// TIA Portal project "Programa_G10" (V18)

(* hardware
DEVICE "S71500/ET200MP station_1"  S7-1500 station
   slot 0: "Perfil soporte_0"  Rack  6ES7 590-1***0-0AA0
   slot 1: "PLC_1"  CPU 1516-3 PN/DP  6ES7 516-3AN01-0AB0  V2.1
      slot 3: "Display de la CPU_1"  6ES7591-1BA00-0AA0
   slot 2: "DI 32x24VDC HF_1"  DI 32x24VDC HF  6ES7 521-1BL00-0AB0  V2.1
   slot 3: "DQ 32x24VDC/0.5A HF_1"  DQ 32x24VDC/0.5A HF  6ES7 522-1BL01-0AB0  V1.0
   slot 4: "AI 8xU/I/RTD/TC ST_1"  AI 8xU/I/RTD/TC ST  6ES7 531-7KF00-0AB0  V2.1
   slot 5: "AQ 4xU/I ST_1"  AQ 4xU/I ST  6ES7 532-5HD00-0AB0  V2.1
*)

// ===== PLC "PLC_1"  CPU 1516-3 PN/DP =====

VAR_GLOBAL   // PLC tag table "Variables generales"
   "X10" AT %M0.0 : Bool;
   "X_PintadoModoCuadricula" AT %M0.1 : Bool;
   "X_PintadoModoNormal" AT %M0.2 : Bool;
   "ON" AT %E4.5 : Bool;
   "rearme" AT %E4.6 : Bool;
   "Seta_emergencia" AT %E4.7 : Bool;
   "X_Emer" AT %M0.3 : Bool;
END_VAR

VAR_GLOBAL   // PLC tag table "Estacion barnizado"
   "EST_BAR_SP_plat_omni" AT %E0.0 : Bool;
   "EST_BAR_pieza_debe_entrar" AT %E0.1 : Bool;
   "EST_BAR_SP_barnizadora_in" AT %E0.2 : Bool;
   "EST_BAR_SP_barnizadora_out" AT %E0.3 : Bool;
   "EST_BAR_SP_pickplace_grabado_in" AT %E0.4 : Bool;
   "EST_BAR_SP_pickplace_grabado_out" AT %E0.5 : Bool;
   "EST_BAR_SP_grabado" AT %E0.6 : Bool;
   "EST_BAR_Meter_Pieza" AT %A0.0 : Bool;
   "Temp_barnizadora" AT %T0 : Timer;
   "EST_BAR_Temp_ruedas_lim" AT %T1 : Timer;
   "EST_BAR_Temp_ruedas_std" AT %T2 : Timer;
   "EST_BAR_error_plat_omni" AT %A0.2 : Bool;
   "EST_BAR_emer_plat_omni" AT %A0.3 : Bool;
   "EST_BAR_stdby_plat_omni" AT %A0.4 : Bool;
   "EST_BAR_es_pieza" AT %E0.7 : Bool;
   "EST_BAR_es_cilindro" AT %E2.2 : Bool;
   "EST_BAR_es_tablero" AT %E1.1 : Bool;
   "EST_BAR_Temp_lim_pieza" AT %T3 : Timer;
   "EST_BAR_Temp_lim_cilindro" AT %T4 : Timer;
   "EST_BAR_Temp_lim_tablero" AT %T5 : Timer;
   "Barnizar_pieza" AT %A0.5 : Bool;
   "Barnizar_cilindro" AT %A0.6 : Bool;
   "Barnizar_tablero" AT %A0.7 : Bool;
   "EST_BAR_error_barnizadora" AT %A1.0 : Bool;
   "EST_BAR_emer_barnizadora" AT %A1.1 : Bool;
   "EST_BAR_stdby_barnizadora" AT %A1.2 : Bool;
   "EST_BAR_Temp_lim_pickplace_mov1" AT %T6 : Timer;
   "EST_BAR_Temp_lim_pickplace_mov2" AT %T7 : Timer;
   "EST_BAR_Temp_lim_pickplace_mov3" AT %T8 : Timer;
   "EST_BAR_Temp_lim_pickplace_mov4" AT %T9 : Timer;
   "EST_BAR_Temp_lim_pickplace_mov5" AT %T10 : Timer;
   "EST_BAR_pickplace_izq" AT %A1.3 : Bool;
   "EST_BAR_pickplace_coger" AT %A1.4 : Bool;
   "EST_BAR_pickplace_centro" AT %A1.5 : Bool;
   "EST_BAR_pickplace_soltar" AT %A1.6 : Bool;
   "EST_BAR_pickplace_ir_a_reposo" AT %A1.7 : Bool;
   "EST_BAR_pickplace_dcha" AT %A2.0 : Bool;
   "EST_BAR_pickplace_EnHome" AT %E1.2 : Bool;
   "EST_BAR_pickplace_EnIzq" AT %E1.3 : Bool;
   "EST_BAR_pickplace_EnCentro" AT %E1.4 : Bool;
   "EST_BAR_pickplace_EnDcha" AT %E1.5 : Bool;
   "EST_BAR_pickplace_pinza_ocupada" AT %E1.6 : Bool;
   "EST_BAR_pickplace_pinza_libre" AT %E1.7 : Bool;
   "EST_BAR_error_pickplace" AT %A2.1 : Bool;
   "EST_BAR_emer_pickplace" AT %A2.2 : Bool;
   "EST_BAR_stdby_pickplace" AT %A2.3 : Bool;
   "EST_BAR_Temp_lim_grabado" AT %T11 : Timer;
   "EST_BAR_Temp_std_grabado" AT %T12 : Timer;
   "EST_BAR_grabar" AT %A2.4 : Bool;
   "EST_BAR_error_grabado" AT %A2.5 : Bool;
   "EST_BAR_emer_grabado" AT %A2.6 : Bool;
   "EST_BAR_stdby_grabado" AT %A2.7 : Bool;
   "EST_BAR_grabado_terminado" AT %E2.3 : Bool;
END_VAR

VAR_GLOBAL   // PLC tag table "Estacion pintado"
   "EST_PIN_SP_plat_omni" AT %E2.0 : Bool;
   "EST_PINT_pieza_debe_entrar" AT %E2.1 : Bool;
   "EST_PIN_SP_pickplace_grabado_in" AT %E2.4 : Bool;
   "EST_PIN_SP_pickplace_grabado_out" AT %E2.5 : Bool;
   "EST_PIN_SP_pickplace_pintado_in" AT %E2.6 : Bool;
   "EST_PIN_SP_pickplace_pintado_out" AT %E2.7 : Bool;
   "EST_PIN_Temp_ruedas_lim" AT %T13 : Timer;
   "EST_PIN_Meter_Pieza" AT %A3.0 : Bool;
   "EST_PIN_error_plat_omni" AT %A3.1 : Bool;
   "EST_PIN_emer_plat_omni" AT %A3.2 : Bool;
   "EST_PIN_stdby_plat_omni" AT %A3.3 : Bool;
   "EST_PIN_SP_PiezaEnMesa" AT %E3.0 : Bool;
   "EST_PIN_SP_LaminaEnMesa" AT %E3.1 : Bool;
   "EST_PIN_SP_LaminaEnPosInicial" AT %E3.2 : Bool;
   "EST_PIN_Pintado_Terminado" AT %E3.3 : Bool;
   "EST_PIN_Hay_Tablero" AT %E3.4 : Bool;
   "EST_PIN_Temp_pintado_ModoLam" AT %T14 : Timer;
   "EST_PIN_Temp_pintado_ModoNormal" AT %T15 : Timer;
   "Pintar" AT %A3.4 : Bool;
   "EST_PIN_error_pintado" AT %A3.5 : Bool;
   "EST_PIN_emer_pintado" AT %A3.6 : Bool;
   "EST_PIN_stdby_pintado" AT %A3.7 : Bool;
   "EST_PIN_Temp_lim_pickplace_mov1" AT %T16 : Timer;
   "EST_PIN_Temp_lim_pickplace_mov2" AT %T17 : Timer;
   "EST_PIN_Temp_lim_pickplace_mov3" AT %T18 : Timer;
   "EST_PIN_Temp_lim_pickplace_mov4" AT %T19 : Timer;
   "EST_PIN_Temp_lim_pickplace_mov5" AT %T20 : Timer;
   "EST_PIN_pickplace_EnHome" AT %E3.5 : Bool;
   "EST_PIN_pickplace_EnIzq" AT %E3.6 : Bool;
   "EST_PIN_pickplace_EnCentro" AT %E3.7 : Bool;
   "EST_PIN_pickplace_EnDcha" AT %E4.0 : Bool;
   "EST_PIN_pickplace_pinza_ocupada" AT %E4.1 : Bool;
   "EST_PIN_pickplace_pinza_libre" AT %E4.2 : Bool;
   "EST_PIN_pickplace_izq" AT %A4.0 : Bool;
   "EST_PIN_pickplace_coger" AT %A4.1 : Bool;
   "EST_PIN_pickplace_centro" AT %A4.2 : Bool;
   "EST_PIN_pickplace_soltar" AT %A4.3 : Bool;
   "EST_PIN_pickplace_ir_a_reposo" AT %A4.4 : Bool;
   "EST_PIN_pickplace_dcha" AT %A4.5 : Bool;
   "EST_PIN_error_pickplace" AT %A4.6 : Bool;
   "EST_PIN_emer_pickplace" AT %A4.7 : Bool;
   "EST_PIN_stdby_pickplace" AT %A5.0 : Bool;
   "EST_PIN_SP_grabado" AT %E4.3 : Bool;
   "EST_PIN_grabado_terminado" AT %E4.4 : Bool;
   "EST_PIN_Temp_lim_grabado" AT %T21 : Timer;
   "EST_PIN_grabar" AT %A5.1 : Bool;
   "EST_PIN_error_grabado" AT %A5.2 : Bool;
   "EST_PIN_emer_grabado" AT %A5.3 : Bool;
   "EST_PIN_stdby_grabado" AT %A5.4 : Bool;
END_VAR

VAR_GLOBAL   // PLC tag table "Estacion secado"
   "EST_SEC_SP_plat_omni" AT %E1.0 : Bool;
   "EST_SEC_pieza_debe_entrar" AT %E5.0 : Bool;
   "EST_SEC_SP_secadora" AT %E5.1 : Bool;
   "EST_SEC_Meter_Pieza" AT %A5.6 : Bool;
   "EST_SEC_Temp_lim_ruedas" AT %T22 : Timer;
   "EST_SEC_error_plat_omni" AT %A5.7 : Bool;
   "EST_SEC_emer_plat_omni" AT %A6.0 : Bool;
   "EST_SEC_stdby_plat_omni" AT %A6.1 : Bool;
   "EST_SEC_secado_terminado" AT %E5.2 : Bool;
   "EST_SEC_Temp_lim_secado" AT %T23 : Timer;
   "Secar" AT %A6.2 : Bool;
   "EST_SEC_error_desecadora" AT %A6.3 : Bool;
   "EST_SEC_emer_desecadora" AT %A6.4 : Bool;
   "EST_SEC_stdby_desecadora" AT %A6.5 : Bool;
   "EST_SEC_SP_grabado" AT %E5.3 : Bool;
   "EST_SEC_grabado_terminado" AT %E5.4 : Bool;
   "EST_SEC_Temp_lim_grabado" AT %T24 : Timer;
   "EST_SEC_grabar" AT %A6.6 : Bool;
   "EST_SEC_error_grabado" AT %A6.7 : Bool;
   "EST_SEC_emer_grabado" AT %A7.0 : Bool;
   "EST_SEC_stdby_grabado" AT %A7.1 : Bool;
END_VAR

VAR_GLOBAL   // PLC tag table "Cinta"
   "vel_cinta_muestreada_bits" AT %EW4 : Int;
   "Temp_cinta" AT %T40 : Timer;
   "Error_cinta" AT %A10.0 : Bool;
   "Motor_cinta" AT %A10.1 : Bool;
   "velocidad_fuera_rango" AT %A10.2 : Bool;
END_VAR

DATA_BLOCK "Datos_produccion"   // DB1
{ S7_Optimized_Access := 'TRUE' }
VERSION : 0.1
   VAR
      t_lim_respuesta_lectura : S5Time := S5T#10s;
      t_lim_plat_omni : S5Time := S5T#60s;
      t_lim_barnizado : S5Time := S5T#10s;
      t_lim_secado : S5Time := S5T#60s;
      t_lim_pickandplace : S5Time := S5T#10s;
      t_lim_robotpintado : S5Time := S5T#10s;
      t_lim_grabado : S5Time := S5T#60s;
      t_lim_cinta : S5Time := S5T#10s;
      max_malas_lecturas : Word := 30;
      t_fugaz_21 : S5Time := S5T#1s;
      t_lim_pintado : S5Time;
      t_lim_barnizado_pieza : S5Time := S5T#30s;
      t_lim_barnizado_cilindro : S5Time := S5T#70s;
      t_lim_barnizado_tablero : S5Time := S5T#100s;
   END_VAR
BEGIN
END_DATA_BLOCK

// folder: Bloques de datos

DATA_BLOCK "Ruedas_omnidireccionales_DB_EST_BAR"   // DB2
{ S7_Optimized_Access := 'TRUE' }
VERSION : 0.1
// stored: InstanceOfName Ruedas_omnidireccionales
"Ruedas_omnidireccionales"
BEGIN
END_DATA_BLOCK

DATA_BLOCK "Maq_barnizado_DB"   // DB3
{ S7_Optimized_Access := 'TRUE' }
VERSION : 0.1
// stored: InstanceOfName Maq_barnizado
"Maq_barnizado"
BEGIN
END_DATA_BLOCK

DATA_BLOCK "Robot_pickandplace_DB_EST_BAR_1"   // DB4
{ S7_Optimized_Access := 'TRUE' }
VERSION : 0.1
// stored: InstanceOfName Robot_pickandplace
"Robot_pickandplace"
BEGIN
END_DATA_BLOCK

DATA_BLOCK "Maq_grabado_DB_EST_BAR"   // DB5
{ S7_Optimized_Access := 'TRUE' }
VERSION : 0.1
// stored: InstanceOfName Maq_grabado
"Maq_grabado"
BEGIN
END_DATA_BLOCK

DATA_BLOCK "Robot_pickandplace_DB_EST_BAR_2"   // DB6
{ S7_Optimized_Access := 'TRUE' }
VERSION : 0.1
// stored: InstanceOfName Robot_pickandplace
"Robot_pickandplace"
BEGIN
END_DATA_BLOCK

DATA_BLOCK "Ruedas_omnidireccionales_DB_EST_PINT"   // DB7
{ S7_Optimized_Access := 'TRUE' }
VERSION : 0.1
// stored: InstanceOfName Ruedas_omnidireccionales
"Ruedas_omnidireccionales"
BEGIN
END_DATA_BLOCK

DATA_BLOCK "Robot_pintado_DB"   // DB8
{ S7_Optimized_Access := 'TRUE' }
VERSION : 0.1
// stored: InstanceOfName Robot_pintado
"Robot_pintado"
BEGIN
END_DATA_BLOCK

DATA_BLOCK "Robot_pickandplace_DB_EST_PINT_1"   // DB9
{ S7_Optimized_Access := 'TRUE' }
VERSION : 0.1
// stored: InstanceOfName Robot_pickandplace
"Robot_pickandplace"
BEGIN
END_DATA_BLOCK

DATA_BLOCK "Maq_grabado_DB_EST_PINT"   // DB10
{ S7_Optimized_Access := 'TRUE' }
VERSION : 0.1
// stored: InstanceOfName Maq_grabado
"Maq_grabado"
BEGIN
END_DATA_BLOCK

DATA_BLOCK "Ruedas_omnidireccionales_DB_EST_SEC"   // DB11
{ S7_Optimized_Access := 'TRUE' }
VERSION : 0.1
// stored: InstanceOfName Ruedas_omnidireccionales
"Ruedas_omnidireccionales"
BEGIN
END_DATA_BLOCK

DATA_BLOCK "Maq_secado_DB"   // DB12
{ S7_Optimized_Access := 'TRUE' }
VERSION : 0.1
// stored: InstanceOfName Maq_secado
"Maq_secado"
BEGIN
END_DATA_BLOCK

DATA_BLOCK "Maq_grabado_DB_EST_SEC"   // DB13
{ S7_Optimized_Access := 'TRUE' }
VERSION : 0.1
// stored: InstanceOfName Maq_grabado
"Maq_grabado"
BEGIN
END_DATA_BLOCK

DATA_BLOCK "Cinta_DB"   // DB14
{ S7_Optimized_Access := 'TRUE' }
VERSION : 0.1
// stored: InstanceOfName Cinta
"Cinta"
BEGIN
END_DATA_BLOCK

// folder: Modos

DATA_BLOCK "Datos_ModoCuadricula"   // DB20
{ S7_Optimized_Access := 'TRUE' }
VERSION : 0.1
   VAR
      t_lim_pintado_ModoCuadricula : S5Time := S5T#100s;
   END_VAR
BEGIN
END_DATA_BLOCK

DATA_BLOCK "Datos_ModoNormal"   // DB21
{ S7_Optimized_Access := 'TRUE' }
VERSION : 0.1
   VAR
      t_lim_pintado_ModoNormal : S5Time := S5T#180s;
   END_VAR
BEGIN
END_DATA_BLOCK

// folder: (top level)

FUNCTION "Celda_barnizado_secado_pintado" : Void   // FC13, STL
{ S7_Optimized_Access := 'TRUE' }
VERSION : 0.1
BEGIN

REGION Network 1: Llamada a las estaciones
         CALL  "Estacion_barnizado";
         CALL  "Estacion_pintado";
         CALL  "Estacion_secado";
END_REGION

REGION Network 2: Llamada a la cinta

         CALL  "Cinta", "Cinta_DB"
         ( vel_cinta_bits        := "vel_cinta_muestreada_bits",
           t_lim_recuperacion    := "Datos_produccion".t_lim_cinta,
           Temp_lim              := "Temp_cinta",
           START                 := "ON",
           error_asincrono       := "Seta_emergencia",
           rearme                := "rearme",
           Act_motor             := "Motor_cinta",
           aviso_vel_fuera_rango := "Error_cinta"
         );
END_REGION

REGION Network 3: Llamada a las FC de emergencia y de modos
         CALL  "Emergencia";
         CALL  "Modos_pintado";
END_REGION
END_FUNCTION

ORGANIZATION_BLOCK "Main"   // OB1, STL, ProgramCycle
TITLE = "Main Program Sweep (Cycle)"
{ S7_Optimized_Access := 'TRUE' }
VERSION : 0.1
   VAR_INPUT
      Initial_Call : Bool;   // Initial call of this OB
      Remanence : Bool;   // =True, if remanent data are available
   END_VAR
BEGIN

REGION Network 1: Llamada a la celda de barnizado, secado y pintado
         CALL  "Celda_barnizado_secado_pintado";
END_REGION
END_ORGANIZATION_BLOCK

ORGANIZATION_BLOCK "Startup"   // OB100, STL, Startup
TITLE = "Complete Restart"
{ S7_Optimized_Access := 'TRUE' }
VERSION : 0.1
   VAR_INPUT
      LostRetentive : Bool;   // True if retentive data are lost
      LostRTC : Bool;   // True if date and time are lost
   END_VAR
BEGIN

REGION Network 1
         SET;
   //    S     "X0"
         S     "X10";
END_REGION
END_ORGANIZATION_BLOCK

// folder: Cinta

FUNCTION_BLOCK "Cinta"   // FB5, STL
{ S7_Optimized_Access := 'TRUE' }
VERSION : 0.1
   VAR_INPUT
      vel_cinta_bits : Int;
      t_lim_recuperacion : S5Time;
      Temp_lim : Timer;
      START : Bool;
      error_asincrono : Bool;
      rearme : Bool;
   END_VAR
   VAR_OUTPUT
      Act_motor : Bool;
      aviso_vel_fuera_rango : Bool;
   END_VAR
   VAR
      X1 : Bool;
      X2 : Bool;
      X_Err_Velocidad : Bool;
      X_Emer : Bool;
      bit_trabajo : Bool;
      vel_fuera_rango : Bool;
   END_VAR
   VAR_TEMP
      ret_val_scale : Word;
      vel_cinta_rpm : Real;
   END_VAR
BEGIN

REGION Network 1: Desconexión
         AN    #START;
         R     #bit_trabajo;
         R     #Act_motor;
         BEC;
END_REGION

REGION Network 2: Conexión
         A     #START;
         FP    #bit_trabajo;

         S     #X1;
         R     #X2;
         R     #X_Err_Velocidad;
END_REGION

REGION Network 3: Llamada a la función SCALE
         O     #X1;
         O     #X2;

         CALL  SCALE
         ( IN      := #vel_cinta_bits,
           HI_LIM  := 10000.0,
           LO_LIM  := 0.0,
           BIPOLAR := false,
           RET_VAL := #ret_val_scale,
           OUT     := #vel_cinta_rpm
         );
         O     #X1;
         O     #X2;
         A(;
         L     #ret_val_scale;
         L     W#16#0008;
         );
         ==I;
         =     #vel_fuera_rango;
END_REGION

REGION Network 4: X1 ->X2
         A     #X1;
         A     #vel_fuera_rango;
         S     #X2;
         R     #X1;
END_REGION

REGION Network 5: Configuración del temporizador
         A     #X2;
         L     #t_lim_recuperacion;
         SS    #Temp_lim;
END_REGION

REGION Network 6: X2-> X_Err_Cinta
         A     #X2;
         A     #Temp_lim;
         S     #X_Err_Velocidad;
         R     #X2;
END_REGION

REGION Network 7: X2 -> X1
         A     #X2;
         AN    #vel_fuera_rango;
         S     #X1;
         R     #X2;
         R     #Temp_lim;
         FR    #Temp_lim;
END_REGION

REGION Network 8: Tratamiento de X1
         A     #X1;
         S     #Act_motor;
END_REGION

REGION Network 9: Activación de X_Emer
         A     #error_asincrono;
         S     #X_Emer;
         R     #X2;
         R     #X_Err_Velocidad;
END_REGION

REGION Network 10: Tratamiento de X_Emer
         A     #X_Emer;
         R     #bit_trabajo;
         R     #aviso_vel_fuera_rango;
         R     #Act_motor;
         R     #Temp_lim;
         FR    #Temp_lim;
END_REGION

REGION Network 11: Rearme tras emergencia
         A     #X_Emer;
         A     #rearme;
         S     #X1;
         R     #X_Emer;
END_REGION

REGION Network 12: Tratamiento de X_Err_Cinta
         A     #X_Err_Velocidad;
         =     #aviso_vel_fuera_rango;
         A     #X_Err_Velocidad;
         R     #Act_motor;
END_REGION

REGION Network 13: Rearme tras error
         A     #X_Err_Velocidad;
         A     #rearme;
         S     #X1;
         R     #X_Err_Velocidad;
END_REGION
END_FUNCTION_BLOCK

// folder: Emergencia

FUNCTION "Emergencia" : Void   // FC3, STL
{ S7_Optimized_Access := 'TRUE' }
VERSION : 0.1
BEGIN

REGION Network 1: Tratamiento de X_EMER
         A     "Seta_emergencia";
         JCN   _TratamientoEmergencia;
   //LLAMADA A LA CINTA
         CALL  "Cinta", "Cinta_DB"
         ( vel_cinta_bits        := ,
           t_lim_recuperacion    := ,
           Temp_lim              := "Temp_cinta",
           START                 := ,
           error_asincrono       := TRUE,
           rearme                := ,
           Act_motor             := "Motor_cinta",
           aviso_vel_fuera_rango := "Error_cinta"
         );


   //LLAMADA A LAS MÁQUNAS Y ROBOTS DE LA ESTACION DE BARNIZADO
         CALL  "Ruedas_omnidireccionales", "Ruedas_omnidireccionales_DB_EST_BAR"
         ( START                          := ,
           SP_plataforma                  := ,
           evento_meter_pieza_en_estacion := ,
           pieza_metida                   := ,
           Temp_lim                       := "EST_BAR_Temp_ruedas_lim",
           tiempo_lim                     := ,
           EMER                           := true,
           rearme                         := ,
           Actuador                       := "EST_BAR_Meter_Pieza",
           aviso_error                    := "EST_BAR_error_plat_omni",
           aviso_emer                     := "EST_BAR_emer_plat_omni",
           aviso_stdby                    := "EST_BAR_stdby_plat_omni"
         );

         CALL  "Maq_barnizado", "Maq_barnizado_DB"
         ( START               := ,
           Sensor_inicio       := ,
           Sensor_fin          := ,
           evento_pieza        := ,
           evento_cilindro     := ,
           evento_tablero      := ,
           Temp_lim_pieza      := ,
           Temp_lim_cilindro   := "EST_BAR_Temp_lim_cilindro",
           Temp_lim_tablero    := "EST_BAR_Temp_lim_tablero",
           tiempo_lim_pieza    := ,
           tiempo_lim_cilindro := ,
           tiempo_lim_tablero  := ,
           EMER                := true,
           rearme              := ,
           Actuador_piezas     := "Barnizar_pieza",
           Actuador_cilindro   := "Barnizar_cilindro",
           Actuador_tablero    := "Barnizar_tablero",
           aviso_error_maq     := "EST_BAR_error_barnizadora",
           aviso_emer_maq      := "EST_BAR_emer_barnizadora",
           aviso_stdby         := "EST_BAR_stdby_barnizadora"
         );

         CALL  "Robot_pickandplace", "Robot_pickandplace_DB_EST_BAR_1"
         ( START             := ,
           emer              := true,
           rearme            := ,
           tiempo_lim        := ,
           Temp_lim_mov1     := "EST_BAR_Temp_lim_pickplace_mov1",
           Temp_lim_mov2     := "EST_BAR_Temp_lim_pickplace_mov2",
           Temp_lim_mov3     := "EST_BAR_Temp_lim_pickplace_mov3",
           Temp_lim_mov4     := "EST_BAR_Temp_lim_pickplace_mov4",
           Temp_lim_mov5     := "EST_BAR_Temp_lim_pickplace_mov5",
           Condicion_inicio  := ,
           Sensor_mov1       := ,
           Pinza_ocupada     := ,
           Sensor_mov3       := ,
           Pinza_libre       := ,
           Sensor_reposo     := ,
           Mov1              := "EST_BAR_pickplace_izq",
           Mov2              := "EST_BAR_pickplace_coger",
           Mov3              := "EST_BAR_pickplace_centro",
           Mov4              := "EST_BAR_pickplace_soltar",
           Mov5              := "EST_BAR_pickplace_ir_a_reposo",
           aviso_error_robot := "EST_BAR_error_pickplace",
           aviso_emer_robot  := "EST_BAR_emer_pickplace",
           aviso_stdby       := "EST_BAR_stdby_pickplace"
         );

         CALL  "Maq_grabado", "Maq_grabado_DB_EST_BAR"
         ( START                := ,
           Sensor_inicio        := ,
           maquina_ha_terminado := ,
           Temp_lim             := "EST_BAR_Temp_lim_grabado",
           tiempo_lim           := ,
           EMER                 := true,
           rearme               := ,
           Actuador             := "EST_BAR_grabar",
           aviso_error_maq      := "EST_BAR_error_grabado",
           aviso_emer_maq       := "EST_BAR_emer_grabado",
           aviso_stdby          := "EST_BAR_stdby_grabado",
           aviso_a_robot        :=
         );


         CALL  "Robot_pickandplace", "Robot_pickandplace_DB_EST_BAR_2"
         ( START             := ,
           emer              := true,
           rearme            := ,
           tiempo_lim        := ,
           Temp_lim_mov1     := "EST_BAR_Temp_lim_pickplace_mov1",
           Temp_lim_mov2     := "EST_BAR_Temp_lim_pickplace_mov2",
           Temp_lim_mov3     := "EST_BAR_Temp_lim_pickplace_mov3",
           Temp_lim_mov4     := "EST_BAR_Temp_lim_pickplace_mov4",
           Temp_lim_mov5     := "EST_BAR_Temp_lim_pickplace_mov5",
           Condicion_inicio  := ,
           Sensor_mov1       := ,
           Pinza_ocupada     := ,
           Sensor_mov3       := ,
           Pinza_libre       := ,
           Sensor_reposo     := ,
           Mov1              := "EST_BAR_pickplace_centro",
           Mov2              := "EST_BAR_pickplace_coger",
           Mov3              := "EST_BAR_pickplace_dcha",
           Mov4              := "EST_BAR_pickplace_soltar",
           Mov5              := "EST_BAR_pickplace_ir_a_reposo",
           aviso_error_robot := "EST_BAR_error_pickplace",
           aviso_emer_robot  := "EST_BAR_emer_pickplace",
           aviso_stdby       := "EST_BAR_stdby_pickplace"
         );



   //LLAMADA A LAS MAQUINAS Y ROBOTS DE LA ESTACION DE PINTADO

         CALL  "Ruedas_omnidireccionales", "Ruedas_omnidireccionales_DB_EST_PINT"
         ( START                          := ,
           SP_plataforma                  := ,
           evento_meter_pieza_en_estacion := ,
           pieza_metida                   := ,
           Temp_lim                       := "EST_PIN_Temp_ruedas_lim",
           tiempo_lim                     := ,
           EMER                           := TRUE,
           rearme                         := ,
           Actuador                       := "EST_PIN_Meter_Pieza",
           aviso_error                    := "EST_PIN_error_plat_omni",
           aviso_emer                     := "EST_PIN_emer_plat_omni",
           aviso_stdby                    := "EST_PIN_stdby_plat_omni"
         );

         CALL  "Robot_pickandplace", "Robot_pickandplace_DB_EST_PINT_1"
         ( START             := ,
           emer              := TRUE,
           rearme            := ,
           tiempo_lim        := ,
           Temp_lim_mov1     := "EST_PIN_Temp_lim_pickplace_mov1",
           Temp_lim_mov2     := "EST_PIN_Temp_lim_pickplace_mov2",
           Temp_lim_mov3     := "EST_PIN_Temp_lim_pickplace_mov3",
           Temp_lim_mov4     := "EST_PIN_Temp_lim_pickplace_mov4",
           Temp_lim_mov5     := "EST_PIN_Temp_lim_pickplace_mov5",
           Condicion_inicio  := ,
           Sensor_mov1       := ,
           Pinza_ocupada     := ,
           Sensor_mov3       := ,
           Pinza_libre       := ,
           Sensor_reposo     := ,
           Mov1              := "EST_PIN_pickplace_izq",
           Mov2              := "EST_PIN_pickplace_coger",
           Mov3              := "EST_PIN_pickplace_centro",
           Mov4              := "EST_PIN_pickplace_soltar",
           Mov5              := "EST_PIN_pickplace_ir_a_reposo",
           aviso_error_robot := "EST_PIN_error_pickplace",
           aviso_emer_robot  := "EST_PIN_emer_pickplace",
           aviso_stdby       := "EST_PIN_stdby_pickplace"
         );

         CALL  "Robot_pintado", "Robot_pintado_DB"
         ( SP_pieza                      := ,
           SP_lamina_mesa                := ,
           SP_lamina_pos_inicial         := ,
           robot_ha_terminado            := ,
           ModoLamina                    := ,
           ModoNormal                    := ,
           t_lim                         := ,
           EMER                          := true,
           rearme                        := ,
           START                         := ,
           Temp_lim_pintado_con_lam      := "EST_PIN_Temp_pintado_ModoLam",
           Temp_lim_pintado_sin_lam      := "EST_PIN_Temp_pintado_ModoNormal",
           Act_pintar                    := "Pintar",
           bde_tiempo                    := "EST_PIN_error_pintado",
           bit_stdby                     := "EST_PIN_stdby_pintado",
           bit_emer                      := "EST_PIN_emer_pintado",
           aviso_a_robot_lamina_a_mesa   := ,
           aviso_a_robot_lamina_a_origen :=
         );

         CALL  "Maq_grabado", "Maq_grabado_DB_EST_PINT"
         ( START                := ,
           Sensor_inicio        := ,
           maquina_ha_terminado := ,
           Temp_lim             := "EST_PIN_Temp_lim_grabado",
           tiempo_lim           := ,
           EMER                 := true,
           rearme               := ,
           Actuador             := "EST_PIN_grabar",
           aviso_error_maq      := "EST_PIN_error_grabado",
           aviso_emer_maq       := "EST_PIN_emer_grabado",
           aviso_stdby          := "EST_PIN_stdby_grabado",
           aviso_a_robot        :=
         );


   //LLAMADA A LAS MÁQUINAS Y ROBOTS DE LA ESTACIÓN DE SECADO

         CALL  "Ruedas_omnidireccionales", "Ruedas_omnidireccionales_DB_EST_SEC"
         ( START                          := ,
           SP_plataforma                  := ,
           evento_meter_pieza_en_estacion := ,
           pieza_metida                   := ,
           Temp_lim                       := "EST_SEC_Temp_lim_ruedas",
           tiempo_lim                     := ,
           EMER                           := true,
           rearme                         := ,
           Actuador                       := "EST_SEC_Meter_Pieza",
           aviso_error                    := "EST_SEC_error_plat_omni",
           aviso_emer                     := "EST_SEC_emer_plat_omni",
           aviso_stdby                    := "EST_SEC_stdby_plat_omni"
         );

         CALL  "Maq_secado", "Maq_secado_DB"
         ( START                := ,
           Sensor_inicio        := ,
           maquina_ha_terminado := ,
           Temp_lim             := "EST_SEC_Temp_lim_secado",
           tiempo_lim           := ,
           EMER                 := true,
           rearme               := ,
           Actuador             := "Secar",
           aviso_error_maq      := "EST_SEC_error_plat_omni",
           aviso_emer_maq       := "EST_SEC_emer_plat_omni",
           aviso_stdby          := "EST_SEC_stdby_plat_omni",
           aviso_a_robot        :=
         );

         CALL  "Maq_grabado", "Maq_grabado_DB_EST_SEC"
         ( START                := ,
           Sensor_inicio        := ,
           maquina_ha_terminado := ,
           Temp_lim             := "EST_SEC_Temp_lim_grabado",
           tiempo_lim           := ,
           EMER                 := true,
           rearme               := ,
           Actuador             := "EST_SEC_grabar",
           aviso_error_maq      := "EST_SEC_error_grabado",
           aviso_emer_maq       := "EST_SEC_emer_grabado",
           aviso_stdby          := "EST_SEC_stdby_grabado",
           aviso_a_robot        :=
         );


   _TratamientoEmergencia:NOP   0;
         A     "Seta_emergencia";
         R     "X_PintadoModoCuadricula";
         R     "X_PintadoModoNormal";

         BEC;
END_REGION

REGION Network 2: Rearme de la celda mediante el pulsador de rearme sin estar la seta activada.
         A     "X_Emer";
         A     "rearme";
         AN    "Seta_emergencia";
         S     "X10";
         R     "X_Emer";
END_REGION
END_FUNCTION

// folder: Estaciones

FUNCTION "Estacion_secado" : Void   // FC2, STL
{ S7_Optimized_Access := 'TRUE' }
VERSION : 0.1
   VAR_TEMP
      aviso_robot_recoger_pieza_secado : Bool;
      aviso_robot_recoger_pieza_grabado : Bool;
   END_VAR
BEGIN

REGION Network 1
         CALL  "Ruedas_omnidireccionales", "Ruedas_omnidireccionales_DB_EST_SEC"
         ( START                          := "ON",
           SP_plataforma                  := "EST_SEC_SP_plat_omni",
           evento_meter_pieza_en_estacion := "EST_SEC_pieza_debe_entrar",
           pieza_metida                   := "EST_SEC_SP_secadora",
           Temp_lim                       := "EST_SEC_Temp_lim_ruedas",
           tiempo_lim                     := "Datos_produccion".t_lim_plat_omni,
           EMER                           := false,
           rearme                         := "rearme",
           Actuador                       := "EST_SEC_Meter_Pieza",
           aviso_error                    := "EST_SEC_error_plat_omni",
           aviso_emer                     := "EST_SEC_emer_plat_omni",
           aviso_stdby                    := "EST_SEC_stdby_plat_omni"
         );

   //Llamada al pick and place para meter la pieza a la máquina de secado

         CALL  "Maq_secado", "Maq_secado_DB"
         ( START                := "ON",
           Sensor_inicio        := "EST_SEC_SP_secadora",
           maquina_ha_terminado := "EST_SEC_secado_terminado",
           Temp_lim             := "EST_SEC_Temp_lim_secado",
           tiempo_lim           := "Datos_produccion".t_lim_secado,
           EMER                 := false,
           rearme               := "rearme",
           Actuador             := "Secar",
           aviso_error_maq      := "EST_SEC_error_plat_omni",
           aviso_emer_maq       := "EST_SEC_emer_plat_omni",
           aviso_stdby          := "EST_SEC_stdby_plat_omni",
           aviso_a_robot        := #aviso_robot_recoger_pieza_secado
         );

   //Llamada al pick and place para mover la pieza de la máquina a la cinta

   //Llamada al pick and place para meter la pieza en la máquina de grabado

         CALL  "Maq_grabado", "Maq_grabado_DB_EST_SEC"
         ( START                := "ON",
           Sensor_inicio        := "EST_SEC_SP_grabado",
           maquina_ha_terminado := "EST_SEC_grabado_terminado",
           Temp_lim             := "EST_SEC_Temp_lim_grabado",
           tiempo_lim           := "Datos_produccion".t_lim_grabado,
           EMER                 := false,
           rearme               := "rearme",
           Actuador             := "EST_SEC_grabar",
           aviso_error_maq      := "EST_SEC_error_grabado",
           aviso_emer_maq       := "EST_SEC_emer_grabado",
           aviso_stdby          := "EST_SEC_stdby_grabado",
           aviso_a_robot        := #aviso_robot_recoger_pieza_grabado
         );

   //Llamada al pick and place para recoger la pieza de la máquina de grabado
END_REGION
END_FUNCTION

FUNCTION "Estacion_barnizado" : Void   // FC4, STL
{ S7_Optimized_Access := 'TRUE' }
VERSION : 0.1
   VAR_TEMP
      aviso_pickplace_quitar_pieza_grabadora : Bool;
   END_VAR
BEGIN

REGION Network 1: Llamada a todas las unidades que forman la estación de barnizado
         CALL  "Ruedas_omnidireccionales", "Ruedas_omnidireccionales_DB_EST_BAR"
         ( START                          := "ON",
           SP_plataforma                  := "EST_BAR_SP_plat_omni",
           evento_meter_pieza_en_estacion := "EST_BAR_pieza_debe_entrar",
           pieza_metida                   := "EST_BAR_SP_barnizadora_in",
           Temp_lim                       := "EST_BAR_Temp_ruedas_lim",
           tiempo_lim                     := "Datos_produccion".t_lim_plat_omni,
           EMER                           := false,
           rearme                         := "rearme",
           Actuador                       := "EST_BAR_Meter_Pieza",
           aviso_error                    := "EST_BAR_error_plat_omni",
           aviso_emer                     := "EST_BAR_emer_plat_omni",
           aviso_stdby                    := "EST_BAR_stdby_plat_omni"
         );


         CALL  "Maq_barnizado", "Maq_barnizado_DB"
         ( START               := "ON",
           Sensor_inicio       := "EST_BAR_SP_barnizadora_in",
           Sensor_fin          := "EST_BAR_SP_barnizadora_out",
           evento_pieza        := "EST_BAR_es_pieza",
           evento_cilindro     := "EST_BAR_es_cilindro",
           evento_tablero      := "EST_BAR_es_tablero",
           Temp_lim_pieza      := "EST_BAR_Temp_lim_pieza",
           Temp_lim_cilindro   := "EST_BAR_Temp_lim_cilindro",
           Temp_lim_tablero    := "EST_BAR_Temp_lim_tablero",
           tiempo_lim_pieza    := "Datos_produccion".t_lim_barnizado_pieza,
           tiempo_lim_cilindro := "Datos_produccion".t_lim_barnizado_cilindro,
           tiempo_lim_tablero  := "Datos_produccion".t_lim_barnizado_tablero,
           EMER                := false,
           rearme              := "rearme",
           Actuador_piezas     := "Barnizar_pieza",
           Actuador_cilindro   := "Barnizar_cilindro",
           Actuador_tablero    := "Barnizar_tablero",
           aviso_error_maq     := "EST_BAR_error_barnizadora",
           aviso_emer_maq      := "EST_BAR_emer_barnizadora",
           aviso_stdby         := "EST_BAR_stdby_barnizadora"
         );



         CALL  "Robot_pickandplace", "Robot_pickandplace_DB_EST_BAR_1"
         ( START             := "ON",
           emer              := FALSE,
           rearme            := "rearme",
           tiempo_lim        := "Datos_produccion".t_lim_pickandplace,
           Temp_lim_mov1     := "EST_BAR_Temp_lim_pickplace_mov1",
           Temp_lim_mov2     := "EST_BAR_Temp_lim_pickplace_mov2",
           Temp_lim_mov3     := "EST_BAR_Temp_lim_pickplace_mov3",
           Temp_lim_mov4     := "EST_BAR_Temp_lim_pickplace_mov4",
           Temp_lim_mov5     := "EST_BAR_Temp_lim_pickplace_mov5",
           Condicion_inicio  := "EST_BAR_SP_pickplace_grabado_in",
           Sensor_mov1       := "EST_BAR_pickplace_EnIzq",
           Pinza_ocupada     := "EST_BAR_pickplace_pinza_ocupada",
           Sensor_mov3       := "EST_BAR_pickplace_EnCentro",
           Pinza_libre       := "EST_BAR_pickplace_pinza_libre",
           Sensor_reposo     := "EST_BAR_pickplace_EnHome",
           Mov1              := "EST_BAR_pickplace_izq",
           Mov2              := "EST_BAR_pickplace_coger",
           Mov3              := "EST_BAR_pickplace_centro",
           Mov4              := "EST_BAR_pickplace_soltar",
           Mov5              := "EST_BAR_pickplace_ir_a_reposo",
           aviso_error_robot := "EST_BAR_error_pickplace",
           aviso_emer_robot  := "EST_BAR_emer_pickplace",
           aviso_stdby       := "EST_BAR_stdby_pickplace"
         );


         CALL  "Maq_grabado", "Maq_grabado_DB_EST_BAR"
         ( START                := "ON",
           Sensor_inicio        := "EST_BAR_SP_grabado",
           maquina_ha_terminado := "EST_BAR_grabado_terminado",
           Temp_lim             := "EST_BAR_Temp_lim_grabado",
           tiempo_lim           := "Datos_produccion".t_lim_grabado,
           EMER                 := false,
           rearme               := "rearme",
           Actuador             := "EST_BAR_grabar",
           aviso_error_maq      := "EST_BAR_error_grabado",
           aviso_emer_maq       := "EST_BAR_emer_grabado",
           aviso_stdby          := "EST_BAR_stdby_grabado",
           aviso_a_robot        := #aviso_pickplace_quitar_pieza_grabadora
         );



         CALL  "Robot_pickandplace", "Robot_pickandplace_DB_EST_BAR_2"
         ( START             := "ON",
           emer              := FALSE,
           rearme            := "rearme",
           tiempo_lim        := "Datos_produccion".t_lim_pickandplace,
           Temp_lim_mov1     := "EST_BAR_Temp_lim_pickplace_mov1",
           Temp_lim_mov2     := "EST_BAR_Temp_lim_pickplace_mov2",
           Temp_lim_mov3     := "EST_BAR_Temp_lim_pickplace_mov3",
           Temp_lim_mov4     := "EST_BAR_Temp_lim_pickplace_mov4",
           Temp_lim_mov5     := "EST_BAR_Temp_lim_pickplace_mov5",
           Condicion_inicio  := #aviso_pickplace_quitar_pieza_grabadora,
           Sensor_mov1       := "EST_BAR_pickplace_EnCentro",
           Pinza_ocupada     := "EST_BAR_pickplace_pinza_ocupada",
           Sensor_mov3       := "EST_BAR_pickplace_EnDcha",
           Pinza_libre       := "EST_BAR_pickplace_pinza_libre",
           Sensor_reposo     := "EST_BAR_pickplace_EnHome",
           Mov1              := "EST_BAR_pickplace_centro",
           Mov2              := "EST_BAR_pickplace_coger",
           Mov3              := "EST_BAR_pickplace_dcha",
           Mov4              := "EST_BAR_pickplace_soltar",
           Mov5              := "EST_BAR_pickplace_ir_a_reposo",
           aviso_error_robot := "EST_BAR_error_pickplace",
           aviso_emer_robot  := "EST_BAR_emer_pickplace",
           aviso_stdby       := "EST_BAR_stdby_pickplace"
         );
END_REGION
END_FUNCTION

FUNCTION "Estacion_pintado" : Void   // FC5, STL
{ S7_Optimized_Access := 'TRUE' }
VERSION : 0.1
   VAR_TEMP
      aviso_pickplace_llevar_lam_a_mesa : Bool;
      aviso_pickplace_llevar_lam_a_origen : Bool;
      aviso_pickplace_quitar_pieza_grabadora : Bool;
   END_VAR
BEGIN

REGION Network 1

         CALL  "Ruedas_omnidireccionales", "Ruedas_omnidireccionales_DB_EST_PINT"
         ( START                          := "ON",
           SP_plataforma                  := "EST_PIN_SP_plat_omni",
           evento_meter_pieza_en_estacion := "EST_PINT_pieza_debe_entrar",
           pieza_metida                   := "EST_PIN_SP_pickplace_pintado_in",
           Temp_lim                       := "EST_PIN_Temp_ruedas_lim",
           tiempo_lim                     := "Datos_produccion".t_lim_plat_omni,
           EMER                           := FALSE,
           rearme                         := "rearme",
           Actuador                       := "EST_PIN_Meter_Pieza",
           aviso_error                    := "EST_PIN_error_plat_omni",
           aviso_emer                     := "EST_PIN_emer_plat_omni",
           aviso_stdby                    := "EST_PIN_stdby_plat_omni"
         );

         CALL  "Robot_pickandplace", "Robot_pickandplace_DB_EST_PINT_1"
         ( START             := "ON",
           emer              := FALSE,
           rearme            := "rearme",
           tiempo_lim        := "Datos_produccion".t_lim_pickandplace,
           Temp_lim_mov1     := "EST_PIN_Temp_lim_pickplace_mov1",
           Temp_lim_mov2     := "EST_PIN_Temp_lim_pickplace_mov2",
           Temp_lim_mov3     := "EST_PIN_Temp_lim_pickplace_mov3",
           Temp_lim_mov4     := "EST_PIN_Temp_lim_pickplace_mov4",
           Temp_lim_mov5     := "EST_PIN_Temp_lim_pickplace_mov5",
           Condicion_inicio  := "EST_PIN_SP_pickplace_pintado_in",
           Sensor_mov1       := "EST_PIN_pickplace_EnIzq",
           Pinza_ocupada     := "EST_PIN_pickplace_pinza_ocupada",
           Sensor_mov3       := "EST_PIN_pickplace_EnCentro",
           Pinza_libre       := "EST_PIN_pickplace_pinza_libre",
           Sensor_reposo     := "EST_PIN_pickplace_EnHome",
           Mov1              := "EST_PIN_pickplace_izq",
           Mov2              := "EST_PIN_pickplace_coger",
           Mov3              := "EST_PIN_pickplace_centro",
           Mov4              := "EST_PIN_pickplace_soltar",
           Mov5              := "EST_PIN_pickplace_ir_a_reposo",
           aviso_error_robot := "EST_PIN_error_pickplace",
           aviso_emer_robot  := "EST_PIN_emer_pickplace",
           aviso_stdby       := "EST_PIN_stdby_pickplace"
         );


         CALL  "Robot_pintado", "Robot_pintado_DB"
         ( SP_pieza                      := "EST_PIN_SP_PiezaEnMesa",
           SP_lamina_mesa                := "EST_PIN_SP_LaminaEnMesa",
           SP_lamina_pos_inicial         := "EST_PIN_SP_LaminaEnPosInicial",
           robot_ha_terminado            := "EST_PIN_Pintado_Terminado",
           ModoLamina                    := "X_PintadoModoNormal",
           ModoNormal                    := "X_PintadoModoCuadricula",
           t_lim                         := "Datos_produccion".t_lim_pintado,
           EMER                          := false,
           rearme                        := "rearme",
           START                         := "ON",
           Temp_lim_pintado_con_lam      := "EST_PIN_Temp_pintado_ModoLam",
           Temp_lim_pintado_sin_lam      := "EST_PIN_Temp_pintado_ModoNormal",
           Act_pintar                    := "Pintar",
           bde_tiempo                    := "EST_PIN_error_pintado",
           bit_stdby                     := "EST_PIN_stdby_pintado",
           bit_emer                      := "EST_PIN_emer_pintado",
           aviso_a_robot_lamina_a_mesa   := #aviso_pickplace_llevar_lam_a_mesa,
           aviso_a_robot_lamina_a_origen := #aviso_pickplace_llevar_lam_a_origen
         );

   //Dos llamadas al pick and place, una para que lleve la lámina del origen a la mesa
   //y otra para que devuelve la lámina de la mesa al lugar donde se encontraba

   //Llamada al pick and place para mover la pieza desde la mesa de pintado hasta la cinta

   //Llamada al pick and place para mover la pieza de la mesa a la máquina de grabado

         CALL  "Maq_grabado", "Maq_grabado_DB_EST_PINT"
         ( START                := "ON",
           Sensor_inicio        := "EST_PIN_SP_grabado",
           maquina_ha_terminado := "EST_PIN_grabado_terminado",
           Temp_lim             := "EST_PIN_Temp_lim_grabado",
           tiempo_lim           := "Datos_produccion".t_lim_grabado,
           EMER                 := false,
           rearme               := "rearme",
           Actuador             := "EST_PIN_grabar",
           aviso_error_maq      := "EST_PIN_error_grabado",
           aviso_emer_maq       := "EST_PIN_emer_grabado",
           aviso_stdby          := "EST_PIN_stdby_grabado",
           aviso_a_robot        := #aviso_pickplace_quitar_pieza_grabadora
         );

   //Llamada al pick and place para que mueva la pieza desde la máquina de grabado hasta la cinta
END_REGION
END_FUNCTION

// folder: Maniobras

FUNCTION_BLOCK "man_simple1_con_err"   // FB1, STL
{ S7_Optimized_Access := 'TRUE' }
VERSION : 0.1
   VAR_INPUT
      sini : Bool;
      sfin : Bool;
      tiempo_lim : S5Time;
      Temp_lim : Timer;
      RESET : Bool;
   END_VAR
   VAR_OUTPUT
      Actuador_man : Bool;
      aviso_error_man : Bool;
      aviso_fin_ok_man : Bool;
   END_VAR
   VAR
      bit_trabajo : Bool;
      X0 : Bool;
      X_Act : Bool;
      X_Fin_Correcto : Bool;
      X_Error_Sincrono : Bool;
   END_VAR
BEGIN

REGION Network 1: Desconexión por RESET
         A     #RESET;
   //Resetar bits
         R     #bit_trabajo;
         R     #aviso_error_man;
         R     #aviso_fin_ok_man;
   //Resetear actuadore
         R     #Actuador_man;
   //Resetear y habilitar temporizador
         R     #Temp_lim;
         FR    #Temp_lim;
         BEC;
END_REGION

REGION Network 2: Desconexión por error síncrono
         A     #X_Error_Sincrono;
         S     #aviso_error_man;
         R     #X_Error_Sincrono;

   //Resetar bits
         R     #bit_trabajo;
         R     #aviso_fin_ok_man;
   //Resetear actuadore
         R     #Actuador_man;
   //Resetear y habilitar temporizador
         R     #Temp_lim;
         FR    #Temp_lim;
         BEC;
END_REGION

REGION Network 3: Desconexión por finalización correcta
         A     #X_Fin_Correcto;
         S     #aviso_fin_ok_man;
         R     #X_Fin_Correcto;

   //Resetar bits
         R     #bit_trabajo;
         R     #aviso_error_man;
   //Resetear actuadore
         R     #Actuador_man;
   //Resetear y habilitar temporizador
         R     #Temp_lim;
         FR    #Temp_lim;
         BEC;
END_REGION

REGION Network 4: Arranque
         SET;
         FP    #bit_trabajo;
         S     #X0;
         R     #X_Act;
         R     #X_Fin_Correcto;
         R     #X_Error_Sincrono;
END_REGION

REGION Network 5: X0 -> X_Error_Sincrono (por mala configuración)
         A     #X0;
         A(;
         ON    #sini;
         O     #sfin;
         );
         S     #X_Error_Sincrono;
         R     #X0;
END_REGION

REGION Network 6: X0-> X_Act
         A     #X0;
         A     #sini;
         S     #X_Act;
         R     #X0;
END_REGION

REGION Network 7: Configuración del perro guardián
         A     #X_Act;
         L     #tiempo_lim;
         SS    #Temp_lim;
END_REGION

REGION Network 8: X_Act -> X_Fin_Correcto
         A     #X_Act;
         A     #sfin;
         S     #X_Fin_Correcto;
         R     #X_Act;
END_REGION

REGION Network 9: Activacion de X_Error_Sincrono (por exceso de tiempo)
         A     #Temp_lim;
         =     #X_Error_Sincrono;
END_REGION

REGION Network 10: Tratamiento de X_Act
         A     #X_Act;
         =     #Actuador_man;
END_REGION
END_FUNCTION_BLOCK

// folder: Modos

FUNCTION "Modos_pintado" : Void   // FC1, STL
TITLE = Grafcet de modos de pintado
{ S7_Optimized_Access := 'TRUE' }
VERSION : 0.1
// Si se activa el sensor de presencia y sensor de lectura detecta un tablero de ajedrez, se activa el pintado modo cuadrícula, que se define en el FB de pintado. Si no, se activa el pintado modo normal.
BEGIN

REGION Network 1: X10 -> X_PintadoModoCuadricula
         A     "X10";
         A     "EST_PIN_SP_PiezaEnMesa";
         A     "EST_PIN_Hay_Tablero";
         S     "X_PintadoModoCuadricula";
         R     "X10";
END_REGION

REGION Network 2: X_PintadoModoCuadricula -> X10
         A     "X_PintadoModoCuadricula";
         A     "EST_PIN_Pintado_Terminado";
         S     "X10";
         R     "X_PintadoModoCuadricula";
END_REGION

REGION Network 3: X10 -> X_PintadoModoNormal
         A     "X10";
         A     "EST_PIN_SP_PiezaEnMesa";
         AN    "EST_PIN_Hay_Tablero";
         S     "X_PintadoModoNormal";
         R     "X10";
END_REGION

REGION Network 4: X_PintadoModoNormal -> X10
         A     "X_PintadoModoNormal";
         A     "EST_PIN_Pintado_Terminado";
         S     "X10";
         R     "X_PintadoModoNormal";
END_REGION

REGION Network 5: Tratamiento de X_PintadoModoCuadricula
         A     "X_PintadoModoCuadricula";
         JCN   _001;
         L     "Datos_ModoCuadricula".t_lim_pintado_ModoCuadricula;
         T     "Datos_produccion".t_lim_pintado;
   _001: NOP   0;
END_REGION

REGION Network 6: Tratamiento de X_PintadoModoNormal
         A     "X_PintadoModoNormal";
         JCN   _002;
         L     "Datos_ModoNormal".t_lim_pintado_ModoNormal;
         T     "Datos_produccion".t_lim_pintado;
   _002: NOP   0;
END_REGION
END_FUNCTION

// folder: Unidades productivas

FUNCTION_BLOCK "Maq_barnizado"   // FB2, STL
{ S7_Optimized_Access := 'TRUE' }
VERSION : 0.1
   VAR_INPUT
      START : Bool;
      Sensor_inicio : Bool;
      Sensor_fin : Bool;
      evento_pieza : Bool;
      evento_cilindro : Bool;
      evento_tablero : Bool;
      Temp_lim_pieza : Timer;
      Temp_lim_cilindro : Timer;
      Temp_lim_tablero : Timer;
      tiempo_lim_pieza : S5Time;
      tiempo_lim_cilindro : S5Time;
      tiempo_lim_tablero : S5Time;
      EMER : Bool;
      rearme : Bool;
   END_VAR
   VAR_OUTPUT
      Actuador_piezas : Bool;
      Actuador_cilindro : Bool;
      Actuador_tablero : Bool;
      aviso_error_maq : Bool;
      aviso_emer_maq : Bool;
      aviso_stdby : Bool;
   END_VAR
   VAR
      man_barnizado_pieza : "man_simple1_con_err";
      man_barnizado_cilindro : "man_simple1_con_err";
      man_barnizado_tablero : "man_simple1_con_err";
      X_Stdby : Bool;
      X2 : Bool;
      X_Man_Pieza : Bool;
      X_Man_Cilindro : Bool;
      X_Man_Tablero : Bool;
      X_Err : Bool;
      X_Emer : Bool;
      bit_trabajo : Bool;
   END_VAR
   VAR_TEMP
      fin_correcto_man_pieza : Bool;
      fin_correcto_man_cilindro : Bool;
      fin_correcto_man_tablero : Bool;
      fin_error_man_pieza : Bool;
      fin_error_man_cilindro : Bool;
      fin_error_man_tablero : Bool;
   END_VAR
BEGIN

REGION Network 1: Desconexión
         AN    #START;
         R     #bit_trabajo;
         R     #aviso_emer_maq;
         R     #aviso_error_maq;

         JCN   _desconectar_maniobras;
         CALL  #man_barnizado_pieza
         ( sini             := ,
           sfin             := ,
           tiempo_lim       := ,
           Temp_lim         := #Temp_lim_pieza,
           RESET            := true,
           Actuador_man     := #Actuador_piezas,
           aviso_error_man  := #fin_correcto_man_pieza,
           aviso_fin_ok_man := #fin_error_man_pieza
         );
         CALL  #man_barnizado_cilindro
         ( sini             := ,
           sfin             := ,
           tiempo_lim       := ,
           Temp_lim         := #Temp_lim_cilindro,
           RESET            := true,
           Actuador_man     := #Actuador_cilindro,
           aviso_error_man  := #fin_correcto_man_cilindro,
           aviso_fin_ok_man := #fin_error_man_cilindro
         );
         CALL  #man_barnizado_tablero
         ( sini             := ,
           sfin             := ,
           tiempo_lim       := ,
           Temp_lim         := #Temp_lim_tablero,
           RESET            := true,
           Actuador_man     := #Actuador_tablero,
           aviso_error_man  := #fin_error_man_tablero,
           aviso_fin_ok_man := #fin_correcto_man_tablero
         );
   _desconectar_maniobras:NOP   0;

         AN    #START;
         BEC;
END_REGION

REGION Network 2: Conexión
         A     #START;
         FP    #bit_trabajo;
         S     #X_Stdby;
         R     #X2;
         R     #X_Man_Pieza;
         R     #X_Man_Cilindro;
         R     #X_Man_Tablero;
         R     #X_Err;
         R     #X_Emer;
END_REGION

REGION Network 3: X_Stdby -> X2
         A     #X_Stdby;
         A     #Sensor_inicio;
         S     #X2;
         R     #X_Stdby;
END_REGION

REGION Network 4: X2-> X_Man_Pieza
         A     #X2;
         A     #evento_pieza;
         S     #X_Man_Pieza;
         R     #X2;
END_REGION

REGION Network 5: X2-> X_Man_Cilindro
         A     #X2;
         A     #evento_cilindro;
         S     #X_Man_Cilindro;
         R     #X2;
END_REGION

REGION Network 6: X2-> X_Man_Tablero
         A     #X2;
         A     #evento_tablero;
         S     #X_Man_Tablero;
         R     #X2;
END_REGION

REGION Network 7: Tratamiento de la maniobra barnizado pieza, X_Man_Pieza -> X_Stdby, X_Man_Pieza -> X_Err
         A     #X_Man_Pieza;
         JCN   _barnizar_pieza;
         CALL  #man_barnizado_pieza
         ( sini             := #Sensor_inicio,
           sfin             := #Sensor_fin,
           tiempo_lim       := #tiempo_lim_pieza,
           Temp_lim         := #Temp_lim_pieza,
           RESET            := false,
           Actuador_man     := #Actuador_piezas,
           aviso_error_man  := #fin_error_man_pieza,
           aviso_fin_ok_man := #fin_correcto_man_pieza
         );
         A     #fin_error_man_pieza;
         S     #X_Err;
         R     #X_Man_Pieza;

         A     #fin_correcto_man_pieza;
         S     #X_Stdby;
         R     #X_Man_Pieza;
   _barnizar_pieza:NOP   0;
END_REGION

REGION Network 8: Tratamiento de la maniobra barnizado cilindro, X_Man_Cilindro -> X_Stdby, X_Man_Cilindro -> X_Err
         A     #X_Man_Cilindro;
         JCN   _barnizar_cilindro;

         CALL  #man_barnizado_cilindro
         ( sini             := #Sensor_inicio,
           sfin             := #Sensor_fin,
           tiempo_lim       := #tiempo_lim_cilindro,
           Temp_lim         := #Temp_lim_cilindro,
           RESET            := false,
           Actuador_man     := #Actuador_cilindro,
           aviso_error_man  := #fin_error_man_cilindro,
           aviso_fin_ok_man := #fin_correcto_man_cilindro
         );

         A     #fin_error_man_cilindro;
         S     #X_Err;
         R     #X_Man_Cilindro;

         A     #fin_correcto_man_cilindro;
         S     #X_Stdby;
         R     #X_Man_Cilindro;

   _barnizar_cilindro:NOP   0;
END_REGION

REGION Network 9: Tratamiento de la maniobra barnizado tablero, X_Man_Tablero -> X_Stdby, X_Man_Tablero -> X_Err
         A     #X_Man_Tablero;
         JCN   _barnizar_tablero;

         CALL  #man_barnizado_tablero
         ( sini             := #Sensor_inicio,
           sfin             := #Sensor_fin,
           tiempo_lim       := #tiempo_lim_tablero,
           Temp_lim         := #Temp_lim_tablero,
           RESET            := false,
           Actuador_man     := #Actuador_tablero,
           aviso_error_man  := #fin_error_man_tablero,
           aviso_fin_ok_man := #fin_correcto_man_tablero
         );

         A     #fin_error_man_tablero;
         S     #X_Err;
         R     #X_Man_Tablero;

         A     #fin_correcto_man_tablero;
         S     #X_Stdby;
         R     #X_Man_Tablero;

   _barnizar_tablero:NOP   0;
END_REGION

REGION Network 10: Tratamiento de X_Err
         A     #X_Err;
         =     #aviso_error_maq;
         JCN   _informar_man_de_error;
         CALL  #man_barnizado_pieza
         ( sini             := ,
           sfin             := ,
           tiempo_lim       := ,
           Temp_lim         := #Temp_lim_pieza,
           RESET            := true,
           Actuador_man     := #Actuador_piezas,
           aviso_error_man  := #fin_correcto_man_pieza,
           aviso_fin_ok_man := #fin_error_man_pieza
         );

         CALL  #man_barnizado_cilindro
         ( sini             := ,
           sfin             := ,
           tiempo_lim       := ,
           Temp_lim         := #Temp_lim_cilindro,
           RESET            := true,
           Actuador_man     := #Actuador_cilindro,
           aviso_error_man  := #fin_correcto_man_cilindro,
           aviso_fin_ok_man := #fin_error_man_cilindro
         );

         CALL  #man_barnizado_tablero
         ( sini             := ,
           sfin             := ,
           tiempo_lim       := ,
           Temp_lim         := #Temp_lim_tablero,
           RESET            := true,
           Actuador_man     := #Actuador_tablero,
           aviso_error_man  := #fin_error_man_tablero,
           aviso_fin_ok_man := #fin_correcto_man_tablero
         );


   _informar_man_de_error:NOP   0;
END_REGION

REGION Network 11: Rearme del error: X_Err -> X_Stdby
         A     #X_Err;
         A     #rearme;
         S     #X_Stdby;
         R     #X_Err;
END_REGION

REGION Network 12: Activación de X_Emer
         A     #EMER;
         S     #X_Emer;
         R     #X_Stdby;
         R     #X_Man_Pieza;
END_REGION

REGION Network 13: Tratamiento de X_Emer
         A     #X_Emer;
         =     #aviso_emer_maq;

         JCN   _informar_man_de_emergencia;
         CALL  #man_barnizado_pieza
         ( sini             := ,
           sfin             := ,
           tiempo_lim       := ,
           Temp_lim         := #Temp_lim_pieza,
           RESET            := true,
           Actuador_man     := #Actuador_piezas,
           aviso_error_man  := #fin_correcto_man_pieza,
           aviso_fin_ok_man := #fin_error_man_pieza
         );

         CALL  #man_barnizado_cilindro
         ( sini             := ,
           sfin             := ,
           tiempo_lim       := ,
           Temp_lim         := #Temp_lim_cilindro,
           RESET            := true,
           Actuador_man     := #Actuador_cilindro,
           aviso_error_man  := #fin_correcto_man_cilindro,
           aviso_fin_ok_man := #fin_error_man_cilindro
         );

         CALL  #man_barnizado_tablero
         ( sini             := ,
           sfin             := ,
           tiempo_lim       := ,
           Temp_lim         := #Temp_lim_tablero,
           RESET            := true,
           Actuador_man     := #Actuador_tablero,
           aviso_error_man  := #fin_error_man_tablero,
           aviso_fin_ok_man := #fin_correcto_man_tablero
         );

   _informar_man_de_emergencia:NOP   0;
END_REGION

REGION Network 14: Rearme del estado de emergencia: X_Emer
         A     #X_Emer;
         A     #rearme;
         S     #X_Stdby;
         R     #X_Emer;
END_REGION

REGION Network 15: Activación del aviso de standby
         A     #X_Stdby;
         =     #aviso_stdby;
END_REGION
END_FUNCTION_BLOCK

FUNCTION_BLOCK "Maq_grabado"   // FB3, STL
{ S7_Optimized_Access := 'TRUE' }
VERSION : 0.1
   VAR_INPUT
      START : Bool;
      Sensor_inicio : Bool;
      maquina_ha_terminado : Bool;
      Temp_lim : Timer;
      tiempo_lim : S5Time;
      EMER : Bool;
      rearme : Bool;
   END_VAR
   VAR_OUTPUT
      Actuador : Bool;
      aviso_error_maq : Bool;
      aviso_emer_maq : Bool;
      aviso_stdby : Bool;
      aviso_a_robot : Bool;
   END_VAR
   VAR
      X_Stdby : Bool;
      X_Man : Bool;
      X_Aviso_Robot : Bool;
      X_Err : Bool;
      X_Emer : Bool;
      bit_trabajo : Bool;
      man_grabado : "man_simple1_con_err";
   END_VAR
   VAR_TEMP
      fin_correcto_man : Bool;
      fin_error_man : Bool;
   END_VAR
BEGIN

REGION Network 1: Desconexión
         AN    #START;
         R     #bit_trabajo;
         R     #aviso_emer_maq;
         R     #aviso_error_maq;
         R     #aviso_a_robot;

         JCN   _desconectar_maniobra;
         CALL  #man_grabado
         ( sini             := ,
           sfin             := ,
           tiempo_lim       := ,
           Temp_lim         := #Temp_lim,
           RESET            := true,
           Actuador_man     := #Actuador,
           aviso_error_man  := #fin_error_man,
           aviso_fin_ok_man := #fin_correcto_man
         );

   _desconectar_maniobra:NOP   0;

         AN    #START;
         BEC;
END_REGION

REGION Network 2: Conexión
         A     #START;
         FP    #bit_trabajo;
         S     #X_Stdby;
         R     #X_Man;
         R     #X_Err;
         R     #X_Emer;
         R     #X_Aviso_Robot;
END_REGION

REGION Network 3: X_Stdby -> X_Man
         A     #X_Stdby;
         A     #Sensor_inicio;
         S     #X_Man;
         R     #X_Stdby;
END_REGION

REGION Network 4: X_Aviso_Robot -> X_Stdby
         A     #X_Aviso_Robot;
         AN    #Sensor_inicio;
         R     #X_Aviso_Robot;
         S     #X_Stdby;
END_REGION

REGION Network 5: Tratamiento de la maniobra, X_Man -> X_Aviso_Robot, X_Man -> X_Err
         A     #X_Man;
         JCN   _llamada_a_maniobra;
         CALL  #man_grabado
         ( sini             := #Sensor_inicio,
           sfin             := #maquina_ha_terminado,
           tiempo_lim       := #tiempo_lim,
           Temp_lim         := #Temp_lim,
           RESET            := false,
           Actuador_man     := #Actuador,
           aviso_error_man  := #fin_error_man,
           aviso_fin_ok_man := #fin_correcto_man
         );
         A     #fin_error_man;
         S     #X_Err;
         R     #X_Man;

         A     #fin_correcto_man;
         S     #X_Aviso_Robot;
         R     #X_Man;
   _llamada_a_maniobra:NOP   0;
END_REGION

REGION Network 6: Tratamiento de X_Err
         A     #X_Err;
         =     #aviso_error_maq;
         JCN   _informar_man_de_error;
         CALL  #man_grabado
         ( sini             := ,
           sfin             := ,
           tiempo_lim       := ,
           Temp_lim         := #Temp_lim,
           RESET            := true,
           Actuador_man     := #Actuador,
           aviso_error_man  := #fin_error_man,
           aviso_fin_ok_man := #fin_correcto_man
         );


   _informar_man_de_error:NOP   0;
END_REGION

REGION Network 7: Rearme del error: X_Err -> X_Stdby
         A     #X_Err;
         A     #rearme;
         S     #X_Stdby;
         R     #X_Err;
END_REGION

REGION Network 8: Activación de X_Emer
         A     #EMER;
         S     #X_Emer;
         R     #X_Stdby;
         R     #X_Man;
         R     #X_Aviso_Robot;
END_REGION

REGION Network 9: Tratamiento de X_Emer
         A     #X_Emer;
         =     #aviso_emer_maq;

         JCN   _informar_man_de_emergencia;
         CALL  #man_grabado
         ( sini             := ,
           sfin             := ,
           tiempo_lim       := ,
           Temp_lim         := #Temp_lim,
           RESET            := true,
           Actuador_man     := #Actuador,
           aviso_error_man  := #fin_error_man,
           aviso_fin_ok_man := #fin_correcto_man
         );

   _informar_man_de_emergencia:NOP   0;
END_REGION

REGION Network 10: Rearme del estado de emergencia: X_Emer
         A     #X_Emer;
         A     #rearme;
         S     #X_Stdby;
         R     #X_Emer;
END_REGION

REGION Network 11: Activación del aviso de standby
         A     #X_Stdby;
         =     #aviso_stdby;
END_REGION

REGION Network 12: Tratamiento de X_Aviso_Robot
         A     #X_Aviso_Robot;
         =     #aviso_a_robot;
END_REGION
END_FUNCTION_BLOCK

FUNCTION_BLOCK "Ruedas_omnidireccionales"   // FB4, STL
{ S7_Optimized_Access := 'TRUE' }
VERSION : 0.1
   VAR_INPUT
      START : Bool;
      SP_plataforma : Bool;
      evento_meter_pieza_en_estacion : Bool;
      pieza_metida : Bool;
      Temp_lim : Timer;
      tiempo_lim : S5Time;
      EMER : Bool;
      rearme : Bool;
   END_VAR
   VAR_OUTPUT
      Actuador : Bool;
      aviso_error : Bool;
      aviso_emer : Bool;
      aviso_stdby : Bool;
   END_VAR
   VAR
      X_Stdby : Bool;
      X_Man : Bool;
      X_Err : Bool;
      X_Emer : Bool;
      bit_trabajo : Bool;
      man_meter_pieza : "man_simple1_con_err";
   END_VAR
   VAR_TEMP
      fin_correcto_man : Bool;
      fin_error_man : Bool;
   END_VAR
BEGIN

REGION Network 1: Desconexión
         AN    #START;
         R     #bit_trabajo;
         R     #aviso_emer;
         R     #aviso_error;

         JCN   _desconectar_maniobra;
         CALL  #man_meter_pieza
         ( sini             := ,
           sfin             := ,
           tiempo_lim       := ,
           Temp_lim         := #Temp_lim,
           RESET            := true,
           Actuador_man     := #Actuador,
           aviso_error_man  := #fin_error_man,
           aviso_fin_ok_man := #fin_correcto_man
         );


   _desconectar_maniobra:NOP   0;

         AN    #START;
         BEC;
END_REGION

REGION Network 2: Conexión
         A     #START;
         FP    #bit_trabajo;
         S     #X_Stdby;
         R     #X_Man;
         R     #X_Err;
         R     #X_Emer;
END_REGION

REGION Network 3: X_Stdby -> X_Man
         A     #X_Stdby;
         A     #SP_plataforma;
         A     #evento_meter_pieza_en_estacion;
         S     #X_Man;
         R     #X_Stdby;
END_REGION

REGION Network 4: Tratamiento de la maniobra, X_Man -> X_Aviso_Robot, X_Man -> X_Err
         A     #X_Man;
         JCN   _llamada_a_maniobra;
         CALL  #man_meter_pieza
         ( sini             := #SP_plataforma,
           sfin             := #pieza_metida,
           tiempo_lim       := #tiempo_lim,
           Temp_lim         := #Temp_lim,
           RESET            := false,
           Actuador_man     := #Actuador,
           aviso_error_man  := #fin_error_man,
           aviso_fin_ok_man := #fin_correcto_man
         );


         A     #fin_error_man;
         S     #X_Err;
         R     #X_Man;

         A     #fin_correcto_man;
         S     #X_Stdby;
         R     #X_Man;

   _llamada_a_maniobra:NOP   0;
END_REGION

REGION Network 5: Tratamiento de X_Err
         A     #X_Err;
         =     #aviso_error;
         JCN   _informar_man_de_error;
         CALL  #man_meter_pieza
         ( sini             := ,
           sfin             := ,
           tiempo_lim       := ,
           Temp_lim         := #Temp_lim,
           RESET            := true,
           Actuador_man     := #Actuador,
           aviso_error_man  := #fin_error_man,
           aviso_fin_ok_man := #fin_correcto_man
         );


   _informar_man_de_error:NOP   0;
END_REGION

REGION Network 6: Rearme del error: X_Err -> X_Stdby
         A     #X_Err;
         A     #rearme;
         S     #X_Stdby;
         R     #X_Err;
END_REGION

REGION Network 7: Activación de X_Emer
         A     #EMER;
         S     #X_Emer;
         R     #X_Stdby;
         R     #X_Man;
END_REGION

REGION Network 8: Tratamiento de X_Emer
         A     #X_Emer;
         =     #aviso_emer;

         JCN   _informar_man_de_emergencia;
         CALL  #man_meter_pieza
         ( sini             := ,
           sfin             := ,
           tiempo_lim       := ,
           Temp_lim         := #Temp_lim,
           RESET            := true,
           Actuador_man     := #Actuador,
           aviso_error_man  := #fin_error_man,
           aviso_fin_ok_man := #fin_correcto_man
         );

   _informar_man_de_emergencia:NOP   0;
END_REGION

REGION Network 9: Rearme del estado de emergencia: X_Emer
         A     #X_Emer;
         A     #rearme;
         S     #X_Stdby;
         R     #X_Emer;
END_REGION

REGION Network 10: Activación del aviso de standby
         A     #X_Stdby;
         =     #aviso_stdby;
END_REGION
END_FUNCTION_BLOCK

FUNCTION_BLOCK "Robot_pintado"   // FB6, STL
{ S7_Optimized_Access := 'TRUE' }
VERSION : 0.1
   VAR_INPUT
      SP_pieza : Bool;
      SP_lamina_mesa : Bool;
      SP_lamina_pos_inicial : Bool;
      robot_ha_terminado : Bool;
      ModoLamina : Bool;
      ModoNormal : Bool;
      t_lim : S5Time;
      EMER : Bool;
      rearme : Bool;
      START : Bool;
      Temp_lim_pintado_con_lam : Timer;
      Temp_lim_pintado_sin_lam : Timer;
   END_VAR
   VAR_OUTPUT
      Act_pintar : Bool;
      bde_tiempo : Bool;
      bit_stdby : Bool;
      bit_emer : Bool;
      aviso_a_robot_lamina_a_mesa : Bool;
      aviso_a_robot_lamina_a_origen : Bool;
   END_VAR
   VAR
      X_Stdby : Bool;
      X2 : Bool;
      X3 : Bool;
      X_Act_Modo_Lam : Bool;
      X5 : Bool;
      X_Act_Modo_Normal : Bool;
      X_Err_Tiempo : Bool;
      X_Emer : Bool;
      bit_trabajo : Bool;
      man_pintado_normal : "man_simple1_con_err";
      man_pintado_lamina : "man_simple1_con_err";
   END_VAR
   VAR_TEMP
      fin_pintado_normal : Bool;
      fin_pintado_lamina : Bool;
      fin_error_pintado_normal : Bool;
      fin_error_pintado_lamina : Bool;
   END_VAR
BEGIN

REGION Network 1: Desconexión por RESET
   // Resetea la FB de pintado, y llama a la FB de instancia de pick and place.
         AN    #START;
         R     #bit_trabajo;
         R     #bde_tiempo;
         R     #bit_stdby;
         R     #bit_emer;
         R     #aviso_a_robot_lamina_a_mesa;
         R     #aviso_a_robot_lamina_a_origen;

         JCN   _reset_maniobras;
         CALL  #man_pintado_lamina
         ( sini             := #SP_pieza,
           sfin             := #robot_ha_terminado,
           tiempo_lim       := #t_lim,
           Temp_lim         := #Temp_lim_pintado_con_lam,
           RESET            := true,
           Actuador_man     := #Act_pintar,
           aviso_error_man  := #fin_error_pintado_lamina,
           aviso_fin_ok_man := #fin_pintado_lamina
         );


         CALL  #man_pintado_normal
         ( sini             := ,
           sfin             := ,
           tiempo_lim       := ,
           Temp_lim         := #Temp_lim_pintado_sin_lam,
           RESET            := true,
           Actuador_man     := #Act_pintar,
           aviso_error_man  := #fin_error_pintado_normal,
           aviso_fin_ok_man := #fin_pintado_normal
         );



   _reset_maniobras:NOP   0;
         AN    #START;
         BEC;
END_REGION

REGION Network 2: Conexión/Arranque de la FB
         A     #START;
         FP    #bit_trabajo;

         R     #bde_tiempo;
         R     #bit_emer;

         S     #X_Stdby;
         R     #X2;
         R     #X3;
         R     #X_Act_Modo_Lam;
         R     #X5;
         R     #X_Act_Modo_Normal;
         R     #X_Err_Tiempo;
         R     #X_Emer;
END_REGION

REGION Network 3: X_Stdby -> X2
         A     #X_Stdby;
         A     #SP_pieza;
         S     #X2;
         R     #X_Stdby;
END_REGION

REGION Network 4: X2 -> X6 (X_Act_Modo_Normal)
   // Pintado normal, es decir, únicamente consta de un robot de pintado que pulveriza spray sobre la pieza.
         A     #X2;
         A     #ModoNormal;
         S     #X_Act_Modo_Normal;
         R     #X2;
END_REGION

REGION Network 5: X2-> X3
         A     #X2;
         A     #ModoLamina;
         S     #X3;
         R     #X2;
END_REGION

REGION Network 6: X3-> X4 (X_Act_Modo_Lam)
         A     #X3;
         A     #SP_lamina_mesa;
         S     #X_Act_Modo_Lam;
         R     #X3;
END_REGION

REGION Network 7: X5-> X_Stdby
         A     #X5;
         A     #SP_lamina_pos_inicial;
         S     #X_Stdby;
         R     #X5;
END_REGION

REGION Network 8: X6 -> X_Stdby y tratamiento de X6
         A     #X_Act_Modo_Normal;
         JCN   _llamar_maniobra_pintado_normal;
         CALL  #man_pintado_normal
         ( sini             := #SP_pieza,
           sfin             := #robot_ha_terminado,
           tiempo_lim       := #t_lim,
           Temp_lim         := #Temp_lim_pintado_sin_lam,
           RESET            := false,
           Actuador_man     := #Act_pintar,
           aviso_error_man  := #fin_error_pintado_normal,
           aviso_fin_ok_man := #fin_pintado_normal
         );

         A     #fin_error_pintado_normal;
         S     #X_Err_Tiempo;
         R     #X_Act_Modo_Normal;

         A     #fin_pintado_normal;
         S     #X_Stdby;
         R     #X_Act_Modo_Normal;

   _llamar_maniobra_pintado_normal:NOP   0;
END_REGION

REGION Network 9: X4-> X5 y tratamiento de X4
         A     #X_Act_Modo_Lam;
         JCN   _llamar_maniobra_pintado_lamina;
         CALL  #man_pintado_lamina
         ( sini             := #SP_pieza,
           sfin             := #robot_ha_terminado,
           tiempo_lim       := #t_lim,
           Temp_lim         := #Temp_lim_pintado_con_lam,
           RESET            := false,
           Actuador_man     := #Act_pintar,
           aviso_error_man  := #fin_error_pintado_lamina,
           aviso_fin_ok_man := #fin_pintado_lamina
         );

         A     #fin_error_pintado_lamina;
         S     #X_Err_Tiempo;
         R     #X_Act_Modo_Lam;

         A     #fin_pintado_lamina;
         S     #X5;
         R     #X_Act_Modo_Lam;

   _llamar_maniobra_pintado_lamina:NOP   0;
END_REGION

REGION Network 10: Desconexión por error síncrono (error de tiempo de la unidad productiva)
         A     #X_Err_Tiempo;
         =     #bde_tiempo;

         JCN   _informar_maniobras_error_sincrono;
         CALL  #man_pintado_lamina
         ( sini             := #SP_pieza,
           sfin             := #robot_ha_terminado,
           tiempo_lim       := #t_lim,
           Temp_lim         := #Temp_lim_pintado_con_lam,
           RESET            := true,
           Actuador_man     := #Act_pintar,
           aviso_error_man  := #fin_error_pintado_lamina,
           aviso_fin_ok_man := #fin_pintado_lamina
         );


         CALL  #man_pintado_normal
         ( sini             := ,
           sfin             := ,
           tiempo_lim       := ,
           Temp_lim         := #Temp_lim_pintado_sin_lam,
           RESET            := true,
           Actuador_man     := #Act_pintar,
           aviso_error_man  := #fin_error_pintado_normal,
           aviso_fin_ok_man := #fin_pintado_normal
         );



   _informar_maniobras_error_sincrono:NOP   0;
END_REGION

REGION Network 11: Rearme del error síncrono
         A     #X_Err_Tiempo;

         A     #rearme;
         R     #X_Err_Tiempo;
         S     #X_Stdby;
END_REGION

REGION Network 12: Activación de X_Emer
         A     #EMER;
         S     #X_Emer;

         R     #X_Stdby;
         R     #X2;
         R     #X3;
         R     #X_Act_Modo_Lam;
         R     #X_Act_Modo_Normal;
         R     #X5;
END_REGION

REGION Network 13: Tratamiento de X_Emer
         A     #X_Emer;
         =     #bit_emer;

         JCN   _informar_maniobras_de_emer;
         CALL  #man_pintado_lamina
         ( sini             := #SP_pieza,
           sfin             := #robot_ha_terminado,
           tiempo_lim       := #t_lim,
           Temp_lim         := #Temp_lim_pintado_con_lam,
           RESET            := true,
           Actuador_man     := #Act_pintar,
           aviso_error_man  := #fin_error_pintado_lamina,
           aviso_fin_ok_man := #fin_pintado_lamina
         );


         CALL  #man_pintado_normal
         ( sini             := ,
           sfin             := ,
           tiempo_lim       := ,
           Temp_lim         := #Temp_lim_pintado_sin_lam,
           RESET            := true,
           Actuador_man     := #Act_pintar,
           aviso_error_man  := #fin_error_pintado_normal,
           aviso_fin_ok_man := #fin_pintado_normal
         );


   _informar_maniobras_de_emer:NOP   0;
END_REGION

REGION Network 14: Rearme desde X_Emer (X_Emer -> X1)
         A     #X_Emer;
         A     #rearme;
         AN    #EMER;
         S     #X_Stdby;
         R     #X_Emer;
END_REGION

REGION Network 15: Activación del bit de standby
         A     #X_Stdby;
         =     #bit_stdby;
END_REGION

REGION Network 16: Tratamiento de X3
         A     #X3;
         =     #aviso_a_robot_lamina_a_mesa;
END_REGION

REGION Network 17: Tratamiento de X5
         A     #X5;
         =     #aviso_a_robot_lamina_a_origen;
END_REGION
END_FUNCTION_BLOCK

FUNCTION_BLOCK "Maq_secado"   // FB9, STL
{ S7_Optimized_Access := 'TRUE' }
VERSION : 0.1
   VAR_INPUT
      START : Bool;
      Sensor_inicio : Bool;
      maquina_ha_terminado : Bool;
      Temp_lim : Timer;
      tiempo_lim : S5Time;
      EMER : Bool;
      rearme : Bool;
   END_VAR
   VAR_OUTPUT
      Actuador : Bool;
      aviso_error_maq : Bool;
      aviso_emer_maq : Bool;
      aviso_stdby : Bool;
      aviso_a_robot : Bool;
   END_VAR
   VAR
      X_Stdby : Bool;
      X_Man : Bool;
      X_Aviso_Robot : Bool;
      X_Err : Bool;
      X_Emer : Bool;
      bit_trabajo : Bool;
      man_secado : "man_simple1_con_err";
   END_VAR
   VAR_TEMP
      fin_correcto_man : Bool;
      fin_error_man : Bool;
   END_VAR
BEGIN

REGION Network 1: Desconexión
         AN    #START;
         R     #bit_trabajo;
         R     #aviso_emer_maq;
         R     #aviso_error_maq;
         R     #aviso_a_robot;

         JCN   _desconectar_maniobra;
         CALL  #man_secado
         ( sini             := ,
           sfin             := ,
           tiempo_lim       := ,
           Temp_lim         := #Temp_lim,
           RESET            := true,
           Actuador_man     := #Actuador,
           aviso_error_man  := #fin_error_man,
           aviso_fin_ok_man := #fin_correcto_man
         );


   _desconectar_maniobra:NOP   0;

         AN    #START;
         BEC;
END_REGION

REGION Network 2: Conexión
         A     #START;
         FP    #bit_trabajo;
         S     #X_Stdby;
         R     #X_Man;
         R     #X_Err;
         R     #X_Emer;
         R     #X_Aviso_Robot;
END_REGION

REGION Network 3: X_Stdby -> X_Man
         A     #X_Stdby;
         A     #Sensor_inicio;
         S     #X_Man;
         R     #X_Stdby;
END_REGION

REGION Network 4: X_Aviso_Robot -> X_Stdby
         A     #X_Aviso_Robot;
         AN    #Sensor_inicio;
         R     #X_Aviso_Robot;
         S     #X_Stdby;
END_REGION

REGION Network 5: Tratamiento de la maniobra, X_Man -> X_Aviso_Robot, X_Man -> X_Err
         A     #X_Man;
         JCN   _llamada_a_maniobra;
         CALL  #man_secado
         ( sini             := #Sensor_inicio,
           sfin             := #maquina_ha_terminado,
           tiempo_lim       := #tiempo_lim,
           Temp_lim         := #Temp_lim,
           RESET            := false,
           Actuador_man     := #Actuador,
           aviso_error_man  := #fin_error_man,
           aviso_fin_ok_man := #fin_correcto_man
         );

         A     #fin_error_man;
         S     #X_Err;
         R     #X_Man;

         A     #fin_correcto_man;
         S     #X_Aviso_Robot;
         R     #X_Man;

   _llamada_a_maniobra:NOP   0;
END_REGION

REGION Network 6: Tratamiento de X_Err
         A     #X_Err;
         =     #aviso_error_maq;
         JCN   _informar_man_de_error;
         CALL  #man_secado
         ( sini             := ,
           sfin             := ,
           tiempo_lim       := ,
           Temp_lim         := #Temp_lim,
           RESET            := true,
           Actuador_man     := #Actuador,
           aviso_error_man  := #fin_error_man,
           aviso_fin_ok_man := #fin_correcto_man
         );

   _informar_man_de_error:NOP   0;
END_REGION

REGION Network 7: Rearme del error: X_Err -> X_Stdby
         A     #X_Err;
         A     #rearme;
         S     #X_Stdby;
         R     #X_Err;
END_REGION

REGION Network 8: Activación de X_Emer
         A     #EMER;
         S     #X_Emer;
         R     #X_Stdby;
         R     #X_Man;
         R     #X_Aviso_Robot;
END_REGION

REGION Network 9: Tratamiento de X_Emer
         A     #X_Emer;
         =     #aviso_emer_maq;

         JCN   _informar_man_de_emergencia;
         CALL  #man_secado
         ( sini             := ,
           sfin             := ,
           tiempo_lim       := ,
           Temp_lim         := #Temp_lim,
           RESET            := true,
           Actuador_man     := #Actuador,
           aviso_error_man  := #fin_error_man,
           aviso_fin_ok_man := #fin_correcto_man
         );


   _informar_man_de_emergencia:NOP   0;
END_REGION

REGION Network 10: Rearme del estado de emergencia: X_Emer
         A     #X_Emer;
         A     #rearme;
         S     #X_Stdby;
         R     #X_Emer;
END_REGION

REGION Network 11: Activación del aviso de standby
         A     #X_Stdby;
         =     #aviso_stdby;
END_REGION

REGION Network 12: Tratamiento de X_Aviso_Robot
         A     #X_Aviso_Robot;
         =     #aviso_a_robot;
END_REGION
END_FUNCTION_BLOCK

FUNCTION_BLOCK "Robot_pickandplace"   // FB10, STL
{ S7_Optimized_Access := 'TRUE' }
VERSION : 0.1
   VAR_INPUT
      START : Bool;
      emer : Bool;
      rearme : Bool;
      tiempo_lim : S5Time;
      Temp_lim_mov1 : Timer;
      Temp_lim_mov2 : Timer;
      Temp_lim_mov3 : Timer;
      Temp_lim_mov4 : Timer;
      Temp_lim_mov5 : Timer;
      Condicion_inicio : Bool;
      Sensor_mov1 : Bool;
      Pinza_ocupada : Bool;
      Sensor_mov3 : Bool;
      Pinza_libre : Bool;
      Sensor_reposo : Bool;
   END_VAR
   VAR_OUTPUT
      Mov1 : Bool;
      Mov2 : Bool;
      Mov3 : Bool;
      Mov4 : Bool;
      Mov5 : Bool;
      aviso_error_robot : Bool;
      aviso_emer_robot : Bool;
      aviso_stdby : Bool;
   END_VAR
   VAR
      X_Stdby : Bool;
      X2 : Bool;
      X3 : Bool;
      X4 : Bool;
      X5 : Bool;
      X6 : Bool;
      X_Emer : Bool;
      X_Err : Bool;
      bit_trabajo : Bool;
      man_mov1 : "man_simple1_con_err";
      man_mov2 : "man_simple1_con_err";
      man_mov3 : "man_simple1_con_err";
      man_mov4 : "man_simple1_con_err";
      man_mov5 : "man_simple1_con_err";
   END_VAR
   VAR_TEMP
      fin_correcto_mov1 : Bool;
      fin_correcto_mov2 : Bool;
      fin_correcto_mov3 : Bool;
      fin_correcto_mov4 : Bool;
      fin_correcto_mov5 : Bool;
      fin_error_mov1 : Bool;
      fin_error_mov2 : Bool;
      fin_error_mov3 : Bool;
      fin_error_mov4 : Bool;
      fin_error_mov5 : Bool;
   END_VAR
BEGIN

REGION Network 1: Desconexión
         AN    #START;
         R     #bit_trabajo;
         R     #aviso_emer_robot;
         R     #aviso_error_robot;

         JCN   _desconectar_maniobra;


   _desconectar_maniobra:NOP   0;
         CALL  #man_mov1
         ( sini             := ,
           sfin             := ,
           tiempo_lim       := ,
           Temp_lim         := #Temp_lim_mov1,
           RESET            := true,
           Actuador_man     := #Mov1,
           aviso_error_man  := #fin_error_mov1,
           aviso_fin_ok_man := #fin_correcto_mov1
         );

         CALL  #man_mov2
         ( sini             := ,
           sfin             := ,
           tiempo_lim       := ,
           Temp_lim         := #Temp_lim_mov2,
           RESET            := true,
           Actuador_man     := #Mov2,
           aviso_error_man  := #fin_error_mov2,
           aviso_fin_ok_man := #fin_correcto_mov2
         );

         CALL  #man_mov3
         ( sini             := ,
           sfin             := ,
           tiempo_lim       := ,
           Temp_lim         := #Temp_lim_mov3,
           RESET            := true,
           Actuador_man     := #Mov3,
           aviso_error_man  := #fin_error_mov3,
           aviso_fin_ok_man := #fin_correcto_mov3
         );

         CALL  #man_mov4
         ( sini             := ,
           sfin             := ,
           tiempo_lim       := ,
           Temp_lim         := #Temp_lim_mov4,
           RESET            := true,
           Actuador_man     := #Mov4,
           aviso_error_man  := #fin_error_mov4,
           aviso_fin_ok_man := #fin_correcto_mov4
         );

         CALL  #man_mov5
         ( sini             := ,
           sfin             := ,
           tiempo_lim       := ,
           Temp_lim         := #Temp_lim_mov5,
           RESET            := true,
           Actuador_man     := #Mov5,
           aviso_error_man  := #fin_error_mov5,
           aviso_fin_ok_man := #fin_correcto_mov5
         );


         AN    #START;
         BEC;
END_REGION

REGION Network 2: Conexión
         A     #START;
         FP    #bit_trabajo;
         S     #X_Stdby;
         R     #X2;
         R     #X3;
         R     #X4;
         R     #X5;
         R     #X6;
         R     #X_Err;
         R     #X_Emer;
END_REGION

REGION Network 3: X_Stdby -> X2
         A     #X_Stdby;
         A     #Condicion_inicio;
         S     #X2;
         R     #X_Stdby;
END_REGION

REGION Network 4: X2-> X3 y tratamiento de X2
         A     #X2;
         JCN   _man_mov1;
         CALL  #man_mov1
         ( sini             := #Condicion_inicio,
           sfin             := #Pinza_ocupada,
           tiempo_lim       := #tiempo_lim,
           Temp_lim         := #Temp_lim_mov1,
           RESET            := false,
           Actuador_man     := #Mov1,
           aviso_error_man  := #fin_error_mov1,
           aviso_fin_ok_man := #fin_correcto_mov1
         );

         A     #fin_error_mov1;
         S     #X_Err;
         R     #X2;

         A     #fin_correcto_mov1;
         R     #X2;
         S     #X3;
   _man_mov1:NOP   0;
END_REGION

REGION Network 5: X3-> X4 y tratamiento de X3
         A     #X3;
         JCN   _man_mov2;
         CALL  #man_mov2
         ( sini             := #Sensor_mov1,
           sfin             := #Pinza_ocupada,
           tiempo_lim       := #tiempo_lim,
           Temp_lim         := #Temp_lim_mov2,
           RESET            := false,
           Actuador_man     := #Mov2,
           aviso_error_man  := #fin_error_mov2,
           aviso_fin_ok_man := #fin_correcto_mov2
         );

         A     #fin_error_mov2;
         S     #X_Err;
         R     #X3;

         A     #fin_correcto_mov2;
         R     #X3;
         S     #X4;
   _man_mov2:NOP   0;
END_REGION

REGION Network 6: X4->X5 y tratamiento X4
         A     #X4;
         JCN   _man_mov3;
         CALL  #man_mov3
         ( sini             := #Pinza_ocupada,
           sfin             := #Sensor_mov3,
           tiempo_lim       := #tiempo_lim,
           Temp_lim         := #Temp_lim_mov3,
           RESET            := false,
           Actuador_man     := #Mov3,
           aviso_error_man  := #fin_error_mov3,
           aviso_fin_ok_man := #fin_correcto_mov3
         );

         A     #fin_error_mov3;
         S     #X_Err;
         R     #X4;

         A     #fin_correcto_mov3;
         R     #X4;
         S     #X5;
   _man_mov3:NOP   0;
END_REGION

REGION Network 7: X5-> X6 y tratamiento de X5
         A     #X5;
         JCN   _man_mov4;
         CALL  #man_mov4
         ( sini             := #Sensor_mov3,
           sfin             := #Pinza_libre,
           tiempo_lim       := #tiempo_lim,
           Temp_lim         := #Temp_lim_mov4,
           RESET            := false,
           Actuador_man     := #Mov4,
           aviso_error_man  := #fin_error_mov4,
           aviso_fin_ok_man := #fin_correcto_mov4
         );

         A     #fin_error_mov4;
         S     #X_Err;
         R     #X5;

         A     #fin_correcto_mov3;
         R     #X5;
         S     #X6;
   _man_mov4:NOP   0;
END_REGION

REGION Network 8: X6-> X_Stdby y tratamiento de X6
         A     #X6;
         JCN   _man_mov5;
         CALL  #man_mov5
         ( sini             := #Pinza_libre,
           sfin             := #Sensor_reposo,
           tiempo_lim       := #tiempo_lim,
           Temp_lim         := #Temp_lim_mov5,
           RESET            := false,
           Actuador_man     := #Mov5,
           aviso_error_man  := #fin_error_mov5,
           aviso_fin_ok_man := #fin_correcto_mov5
         );

         A     #fin_error_mov5;
         S     #X_Err;
         R     #X6;

         A     #fin_correcto_mov5;
         S     #X_Stdby;
         R     #X6;

   _man_mov5:NOP   0;
END_REGION

REGION Network 9: Tratamiento de X_Err
         A     #X_Err;
         =     #aviso_error_robot;
         JCN   _informar_man_de_error;
         CALL  #man_mov1
         ( sini             := ,
           sfin             := ,
           tiempo_lim       := ,
           Temp_lim         := #Temp_lim_mov1,
           RESET            := true,
           Actuador_man     := #Mov1,
           aviso_error_man  := #fin_error_mov1,
           aviso_fin_ok_man := #fin_correcto_mov1
         );

         CALL  #man_mov2
         ( sini             := ,
           sfin             := ,
           tiempo_lim       := ,
           Temp_lim         := #Temp_lim_mov2,
           RESET            := true,
           Actuador_man     := #Mov2,
           aviso_error_man  := #fin_error_mov2,
           aviso_fin_ok_man := #fin_correcto_mov2
         );

         CALL  #man_mov3
         ( sini             := ,
           sfin             := ,
           tiempo_lim       := ,
           Temp_lim         := #Temp_lim_mov3,
           RESET            := true,
           Actuador_man     := #Mov3,
           aviso_error_man  := #fin_error_mov3,
           aviso_fin_ok_man := #fin_correcto_mov3
         );

         CALL  #man_mov4
         ( sini             := ,
           sfin             := ,
           tiempo_lim       := ,
           Temp_lim         := #Temp_lim_mov4,
           RESET            := true,
           Actuador_man     := #Mov3,
           aviso_error_man  := #fin_error_mov4,
           aviso_fin_ok_man := #fin_correcto_mov4
         );

         CALL  #man_mov5
         ( sini             := ,
           sfin             := ,
           tiempo_lim       := ,
           Temp_lim         := #Temp_lim_mov5,
           RESET            := true,
           Actuador_man     := #Mov5,
           aviso_error_man  := #fin_error_mov5,
           aviso_fin_ok_man := #fin_correcto_mov5
         );


   _informar_man_de_error:NOP   0;
END_REGION

REGION Network 10: Rearme del error: X_Err -> X_Stdby
         A     #X_Err;
         A     #rearme;
         S     #X_Stdby;
         R     #X_Err;
END_REGION

REGION Network 11: Activación de X_Emer
         A     #emer;
         S     #X_Emer;
         R     #X_Stdby;
         R     #X2;
         R     #X3;
         R     #X4;
         R     #X5;
         R     #X6;
END_REGION

REGION Network 12: Tratamiento de X_Emer
         A     #X_Emer;
         =     #aviso_emer_robot;

         JCN   _informar_man_de_emergencia;
         CALL  #man_mov1
         ( sini             := ,
           sfin             := ,
           tiempo_lim       := ,
           Temp_lim         := #Temp_lim_mov1,
           RESET            := true,
           Actuador_man     := #Mov1,
           aviso_error_man  := #fin_error_mov1,
           aviso_fin_ok_man := #fin_correcto_mov1
         );

         CALL  #man_mov2
         ( sini             := ,
           sfin             := ,
           tiempo_lim       := ,
           Temp_lim         := #Temp_lim_mov2,
           RESET            := true,
           Actuador_man     := #Mov2,
           aviso_error_man  := #fin_error_mov2,
           aviso_fin_ok_man := #fin_correcto_mov2
         );

         CALL  #man_mov3
         ( sini             := ,
           sfin             := ,
           tiempo_lim       := ,
           Temp_lim         := #Temp_lim_mov3,
           RESET            := true,
           Actuador_man     := #Mov3,
           aviso_error_man  := #fin_error_mov3,
           aviso_fin_ok_man := #fin_correcto_mov3
         );

         CALL  #man_mov4
         ( sini             := ,
           sfin             := ,
           tiempo_lim       := ,
           Temp_lim         := #Temp_lim_mov4,
           RESET            := true,
           Actuador_man     := #Mov3,
           aviso_error_man  := #fin_error_mov4,
           aviso_fin_ok_man := #fin_correcto_mov4
         );

         CALL  #man_mov5
         ( sini             := ,
           sfin             := ,
           tiempo_lim       := ,
           Temp_lim         := #Temp_lim_mov5,
           RESET            := true,
           Actuador_man     := #Mov5,
           aviso_error_man  := #fin_error_mov5,
           aviso_fin_ok_man := #fin_correcto_mov5
         );

   _informar_man_de_emergencia:NOP   0;
END_REGION

REGION Network 13: Rearme del estado de emergencia: X_Emer
         A     #X_Emer;
         A     #rearme;
         S     #X_Stdby;
         R     #X_Emer;
END_REGION

REGION Network 14: Activación del aviso de standby
         A     #X_Stdby;
         =     #aviso_stdby;
END_REGION
END_FUNCTION_BLOCK